# EPICS substitutions: vacuum/MAIN_TRUNK/db/su1td_agilent4uhv.substitutions
# Agilent4UHV substitutions file

file db/agilent4uhv.db
{
     pattern {LOCA,			DEV,		PORT,		ADDR,	TIMEOUT}
     		 {SBTL,			SU1TD,		4uhv_1,		0,		0.2}
}
file db/agilent4uhv_alias.db
{
     pattern {LOCA,			DEV,		SUB1,					SUB2,					SUB3,						SUB4,				PORT,	ADDR,	TIMEOUT}
     		 {SBTL,			SU1TD,	VDR:IP01:SIP30,		Empty,		VTUS:IP03:SIP30,			VTUS:IP04:SIP30,	4uhv_1,	0,		0.2}
}
